// This function has been automatically generated from the project information.
{attribute 'signature_flag' := '1073741824'}
{attribute 'TcGenerated'}
{attribute 'no-analysis'}
FUNCTION F_GetCompany : WSTRING
VAR_INPUT
	
END_VAR

F_GetCompany := "ekvip automation GmbH";

END_FUNCTION

(* stored: Version 1.1.0.1, ProductVersion 3.1.4026.11
   POU F_GetCompany: Id {bf850028-63ee-4361-907f-6f2008ca9f57}, SpecialFunc None *)
